Fanuc KAREL source: kb00052.KL

-- PROVISIONAL review KL for V940-1; original PC SHA256 5e3336c844adbc2659d1cbf14a7097f8e697ab34a7721beb2bb6ff5aab84ec9e
-- Incomplete behavior may be omitted. Consult companion uncertainty JSON. Do not deploy.
PROGRAM KB00052
%NOLOCKGROUP
VAR
  P1 : INTEGER
  P2 : INTEGER
-- UNRESOLVED_DECL RESULT type=000106
BEGIN
  -- V9_ZERO_TABLE_METADATA_HINT layout=0001; no indexed target words; source/name/runtime held
  -- UNRESOLVED_PC offsets 5-12; opcodes 9D,23
  -- UNRESOLVED_PC offsets 17-24; opcodes 9D,23
  -- UNRESOLVED_PC offsets 29-58; opcodes 27,22,22,27,9D,76,7E,4A
  -- UNRESOLVED_PC offsets 63-67; opcodes 7F
END KB00052
